TYPE ST_StartPathData :
STRUCT
	sObjectID					: STRING := 'MAIN.fbMMServer';
	sMethodID					: STRING := 'MAIN.fbMMServer#M_StartPath';
	iStatus						: INT;
	iNoOfInputArgs				: BYTE := 1;
	iNoOfOutputArgs				: BYTE := 2;
	stInput						: ST_StartPathDataIn;
	stOutput					: ST_StartPathDataOut;	
END_STRUCT
END_TYPE

(* stored: Version 1.1.0.1, ProductVersion 3.1.4024.5
   DUT ST_StartPathData: Id {55588b6e-0b9c-4b0c-b938-d78eb293dce6} *)
